// TIA Portal project "ContadoresCTUCTDCTUD" (V14)
// Trabalho com contadores

(* hardware
DEVICE "S7-1200 station_1"  S7-1200 Station
   slot 0: "Rack_0"  S7-1200 Rack  Rack  V1.0
   slot 1: "PLC_1_contatores"  CPU 1214C DC/DC/DC  6ES7 214-1AG40-0XB0  V4.2
*)

// ===== PLC "PLC_1_contatores"  CPU 1214C DC/DC/DC =====

VAR_GLOBAL   // PLC tag table "Default tag table"
   "System_Byte" AT %MB1 : Byte;
   "FirstScan" AT %M1.0 : Bool;
   "DiagStatusUpdate" AT %M1.1 : Bool;
   "AlwaysTRUE" AT %M1.2 : Bool;
   "AlwaysFALSE" AT %M1.3 : Bool;
   "Clock_Byte" AT %MB0 : Byte;
   "Clock_10Hz" AT %M0.0 : Bool;
   "Clock_5Hz" AT %M0.1 : Bool;
   "Clock_2.5Hz" AT %M0.2 : Bool;
   "Clock_2Hz" AT %M0.3 : Bool;
   "Clock_1.25Hz" AT %M0.4 : Bool;
   "Clock_1Hz" AT %M0.5 : Bool;
   "Clock_0.625Hz" AT %M0.6 : Bool;
   "Clock_0.5Hz" AT %M0.7 : Bool;
   "Tag_1" AT %M10.0 : Bool;
   "Tag_2" AT %M10.1 : Bool;
   "Tag_3" AT %M10.2 : Bool;
   "Tag_4" AT %M11.1 : Bool;
   "Tag_5" AT %M100.1 : Bool;
   "Tag_6" AT %M100.2 : Bool;
   "Tag_7" AT %M100.3 : Bool;
   "Tag_8" AT %M100.4 : Bool;
   "Tag_9" AT %M200.0 : Bool;
   "Tag_10" AT %M200.1 : Bool;
   "Tag_11" AT %M200.2 : Bool;
   "Tag_12" AT %M200.3 : Bool;
   "Tag_13" AT %M200.4 : Bool;
END_VAR

// folder: System blocks/Program resources

DATA_BLOCK "IEC_Counter_0_DB"   // DB1
{ S7_Optimized_Access := 'TRUE' }
AUTHOR : Simatic
FAMILY : IEC
NAME : CNTR
VERSION : 1.0
// stored: InstanceOfName IEC_COUNTER
"IEC_COUNTER"
BEGIN
END_DATA_BLOCK

DATA_BLOCK "IEC_Counter_0_DB_1"   // DB2
{ S7_Optimized_Access := 'TRUE' }
AUTHOR : Simatic
FAMILY : IEC
NAME : CNTR
VERSION : 1.0
// stored: InstanceOfName IEC_COUNTER
"IEC_COUNTER"
BEGIN
END_DATA_BLOCK

DATA_BLOCK "IEC_Counter_0_DB_2"   // DB3
{ S7_Optimized_Access := 'TRUE' }
AUTHOR : Simatic
FAMILY : IEC
NAME : CNTR
VERSION : 1.0
// stored: InstanceOfName IEC_COUNTER
"IEC_COUNTER"
BEGIN
END_DATA_BLOCK

// folder: (top level)

FUNCTION "Contadores" : Void   // FC1, LAD
{ S7_Optimized_Access := 'TRUE' }
VERSION : 0.1
BEGIN

REGION Network 1: CTU
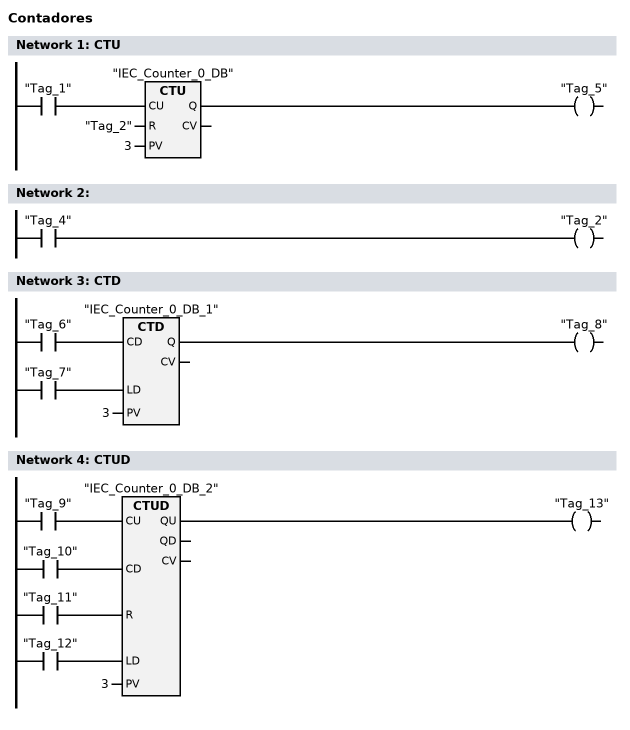
   "IEC_Counter_0_DB".CTU(CU := "Tag_1", R := "Tag_2", PV := 3);
   "Tag_5" := "IEC_Counter_0_DB".Q;
END_REGION

REGION Network 2
   RUNG wire#powerrail
      Contact( "Tag_4" )
      Coil( "Tag_2" )
   END_RUNG
   // the same network as SCL:
   "Tag_2" := "Tag_4";
END_REGION

REGION Network 3: CTD
   "IEC_Counter_0_DB_1".CTD(CD := "Tag_6", LD := "Tag_7", PV := 3);
   "Tag_8" := "IEC_Counter_0_DB_1".Q;
END_REGION

REGION Network 4: CTUD
   "IEC_Counter_0_DB_2".CTUD(CU := "Tag_9", CD := "Tag_10", R := "Tag_11", LD := "Tag_12", PV := 3);
   "Tag_13" := "IEC_Counter_0_DB_2".QU;
END_REGION
END_FUNCTION

ORGANIZATION_BLOCK "Main"   // OB1, LAD, ProgramCycle
TITLE = "Main Program Sweep (Cycle)"
{ S7_Optimized_Access := 'TRUE' }
VERSION : 0.1
   VAR_INPUT
      Initial_Call : Bool;   // Initial call of this OB
      Remanence : Bool;   // =True, if remanent data are available
   END_VAR
BEGIN

REGION Network 1
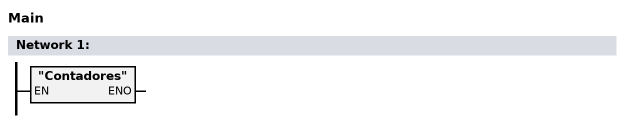
   RUNG wire#powerrail
      "Contadores"()
   END_RUNG
   // the same network as SCL:
   "Contadores"();
END_REGION
END_ORGANIZATION_BLOCK